FUNCTION_BLOCK Hexapod_Leg
VAR_INPUT
	Axis1, Axis2, Axis3	: Axis;
END_VAR
VAR_OUTPUT
END_VAR
VAR
	Axis_Leg		: ARRAY [1..3] OF Axis;
	Axis_Number		: INT;
	Axis_HomeDone	: ARRAY [1..3] OF BOOL;
	HomeDone		: BOOL;
END_VAR

Axis_Leg[1] := Axis1;
Axis_Leg[2] := Axis2;
Axis_Leg[3] := Axis3;

METHOD Home
VAR_INPUT
	Axis1_HomeSet	: BOOL;
	Axis2_HomeSet	: BOOL;
	Axis3_HomeSet	: BOOL;
END_VAR
VAR_OUTPUT	
END_VAR
VAR
	Axis_HomeSet	: BOOL;
END_VAR
IF Axis_HomeDone[1] AND Axis_HomeDone[2] AND Axis_HomeDone[2] THEN
	HomeDone := TRUE;
END_IF

Axis_HomeDone[1] := Axis1.State_HomeDone;
Axis_HomeDone[2] := Axis2.State_HomeDone;
Axis_HomeDone[3] := Axis3.State_HomeDone;
END_METHOD

PROPERTY State_HomeDone : BOOL
GET
State_HomeDone := HomeDone;
END_GET
END_PROPERTY

END_FUNCTION_BLOCK

(* stored: Version 1.1.0.1, ProductVersion 3.1.4020.12
   POU Hexapod_Leg: Id {914f4208-f619-4b5d-a17f-3e0ef39ade98}, SpecialFunc None
   Method Home: Id {959bb286-169d-4f39-a185-0b167baf5e13}
   Property State_HomeDone: Id {7ea31a18-09aa-43dc-a272-2cac98bc6ca4}
   Get Get: Id {d0d12854-8f04-4eb3-8619-591b17832620} *)
